FUNCTION F_Theta_m3 : REAL
VAR_INPUT
END_VAR
VAR
	Pm3 : REAL;
	Pm2: REAL;
	Pm1: REAL;
	Theta0 : REAL:=0;
END_VAR



//Pm3 = mono grating pitch - 63300 urad
Pm3 := Main.M7.fPosition - 63300;

//Pm2 = mono mirror pitch - 90700 urad
Pm2 := Main.M6.fPosition - 90700;

//Pm1 = 18310 - 281 + mr1k1 bend pitch 
Pm1 := 18310 - 281 + Main.M16.fPosition;

F_Theta_m3 := 2 *Pm3 - 2 * Pm2 + 2* Pm1 - Theta0;

END_FUNCTION

(* stored: Version 1.1.0.1, ProductVersion 3.1.4022.12
   POU F_Theta_m3: Id {e2a5921a-7e31-4dc3-8302-5ad55f4155fe}, SpecialFunc None *)
